// TwinCAT 3 PLC project SYNC
// ProgramVersion: 3.1.4022.2
// libraries:
//   Tc2_EtherCAT, * (Beckhoff Automation GmbH)
//   Tc2_MC2, * (Beckhoff Automation GmbH)
//   Tc2_MC2_Camming, * (Beckhoff Automation GmbH)
//   Tc2_MC2_XFC, * (Beckhoff Automation GmbH)
//   Tc2_Standard, * (Beckhoff Automation GmbH)
//   Tc2_System, * (Beckhoff Automation GmbH)
//   Tc3_Module, * (Beckhoff Automation GmbH)
// project tree:
//   / Plc_Task_SYNC.TcTTO
//   POUs/ AxisController.TcPOU, BlockerController.TcPOU, CamInController.TcPOU, MAIN.TcPOU, MODULO.TcPOU
// (motion and I/O tree: see PLC project clock)
// real-time tasks:
//   TASK Plc_Task_CLOCK: cycle T#1ms, priority 20, ADS port 350
//   TASK Plc_Task_SYNC: cycle T#10ms, priority 21, ADS port 351
// variable links:
//   CLOCK Instance <-> SYNC/SYNC Instance
//     PlcTask Outputs/MAIN.tPulse <-> Plc_Task_SYNC Inputs/MAIN.tPulse

CONFIGURATION SYNC
    RESOURCE PLC ON TwinCAT3
        TASK Plc_Task_SYNC(INTERVAL := T#10ms, PRIORITY := 21);
        PROGRAM MAIN WITH Plc_Task_SYNC : MAIN;
    END_RESOURCE
END_CONFIGURATION

// ---- POUs/MAIN.TcPOU
PROGRAM MAIN
VAR
	
	tPulse AT %I*: T_DCTIME64;
	tPrev : T_DCTIME64;
	tPrevPulse : T_DCTIME64;
	tDiff : T_DCTIME64;
	
	SyncMaster : AXIS_REF;
	SyncSlave : AXIS_REF;

	XFC_Position : XFC_PositionAtTime;
	
	fPosition : LREAL;
	fPositionMod : LREAL;
	fPrevPosition : LREAL;
	
	fPositionError : LREAL;
	fPositionSum : LREAL;
	
	fSpeedError : LREAL;
	fSpeedAct : LREAL;
	fSpeed : LREAL := 360*14;
	
	fPositionDiff : LREAL;
	
	Master : AxisController;
	Slave : CamInController;
	
	mcMoveVelo : MC_MoveVelocity;
	
	iState : UINT;
	bPulse : BOOL;
	
	fSpeed_Kp : LREAL := 0.1;
	
	fPosition_Kp : LREAL := 0.1;
	fPosition_Ki : LREAL := 0.001;
	
	fPositionControlThreshold: LREAL := 10;
	
END_VAR

Master(Axis:=SyncMaster);
Master.bExecute:=FALSE;

Slave(Axis:=SyncSlave, Master:=SyncMaster);
Slave.bExecute:=FALSE;

mcMoveVelo(Axis:=SyncMaster);
mcMoveVelo.Execute := FALSE;

CASE iState OF
	000:
		// Compose a camming table?
		
		iState := 100;

	100:
		// Set up the master axis
		Master.fSpeed:=0;
		Master.bExecute := TRUE;
		iState := 101;
	101:
		IF Master.bDone THEN
			iState:= 200;
		END_IF
		
	200:
		// Check for new pulse
		IF tPulse <> tPrev THEN
			// There's a new pusle
			fPrevPosition := fPosition;
			tPrevPulse := tPrev;
			bPulse := TRUE;
		
			// Get the position at the pulse
			XFC_Position(DcTime:=ULINT_TO_UDINT(tPulse), Axis:= SyncMaster);
			fPosition := XFC_Position.Position;
			fPositionMod := MODULO(XFC_Position.Position+180, 360)-180;
			
			// Calculate the distance moved
			fPositionDiff := fPosition-fPrevPosition;
			
			// Calculate the time between pulses
			tDiff := tPulse - tPrevPulse;
			
			// Calculate the actual speed
			fSpeedAct := fPositionDiff/tDiff*1E9;
			
			// Calculate the speed difference - with respect to the expected 360degrees
			fSpeedError := -(fPositionDiff-360)/tDiff*1E9;
			
			// Implement the speed PI controller
			fSpeed := fSpeed + fSpeedError*fSpeed_Kp;
			
			// Implement the position PI controller
			fPositionError := MODULO(fPosition+180, 360)-180;
			fPositionSum := fPositionSum + fPositionError;
			
			// Only activate position control if the speed control is good
			IF ABS(fSpeedError) < fPositionControlThreshold THEN
				fSpeed := fSpeed - fPositionError * fPosition_Kp;
				fSpeed := fSpeed - fPositionSum * fPosition_Ki;
			ELSE
				fPositionSum := 0;
			END_IF
			
			IF fSpeed > 5700 THEN
				fSpeed := 5700;
			END_IF
			
			// Update the velocity
			mcMoveVelo.Execute:= TRUE;
			mcMoveVelo.Velocity:= fSpeed;
			
			(*// Activate slave camming?
			IF NOT Slave.bDone THEN
				Slave.bExecute:=TRUE;
			END_IF*)
		
		ELSE
			bPulse := FALSE;
		END_IF
		
		tPrev := tPulse;
			
END_CASE

END_PROGRAM

// ---- POUs/AxisController.TcPOU
FUNCTION_BLOCK AxisController
VAR_INPUT
	bExecute: BOOL;
	fSpeed : LREAL := 360;
END_VAR
VAR
	mcReset			: MC_Reset;
	mcPower			: MC_Power;
	mcMoveVelo		: MC_MoveVelocity;
	mcStop			: MC_Stop;
	
	iState: UINT;;
END_VAR
VAR_IN_OUT
	Axis : AXIS_REF;
END_VAR
VAR_OUTPUT
	bDone : BOOL;
END_VAR

mcReset(Axis:=Axis);
mcReset.Execute := FALSE;

mcPower(Axis:=Axis, Enable:=TRUE, Enable_Positive:=TRUE, Enable_Negative:=TRUE);

mcMoveVelo(Axis:=Axis);
mcMoveVelo.Execute := FALSE;

CASE iState OF
	0:		
		IF bExecute THEN
			iState:= 10;
		END_IF
		
	10: 
		// Reset the axis
		mcReset.Execute:=TRUE;
		iState := 20;
		bDone:= FALSE;
	
	20: 
		// Wait for reset to complete
		IF McReset.Done THEN
			iState := 30;
		ELSIF McReset.Error THEN
			iState := 999;
		END_IF
	
	30:
		// Set the power!
		IF McPower.Status THEN
			iState := 40;
		END_IF
		
	40: 
		// Move at constant velo
		mcMoveVelo.Execute := TRUE;
		mcMoveVelo.Velocity:=fSpeed;
		
		iState:= 50;
	
	50: 
		// Done.
		IF mcMoveVelo.InVelocity THEN
			bDone := TRUE;
			iState := 0;
		END_IF
		
END_CASE

END_FUNCTION_BLOCK

// ---- POUs/CamInController.TcPOU
FUNCTION_BLOCK CamInController
VAR_INPUT
	bExecute: BOOL;
	fSpeed : LREAL := 360;
END_VAR
VAR
	mcReset			: MC_Reset;
	mcPower			: MC_Power;
	mcStop			: MC_Stop;
	mcCamIn         : MC_CamIn;
	
	iState: UINT;;
END_VAR
VAR_IN_OUT
	Axis : AXIS_REF;
	Master : AXIS_REF;
END_VAR
VAR_OUTPUT
	bDone : BOOL;
END_VAR

mcReset(Axis:=Axis);
mcReset.Execute := FALSE;

mcPower(Axis:=Axis, Enable:=TRUE, Enable_Positive:=TRUE, Enable_Negative:=TRUE);

mcCamIn(Slave:=Axis, Master:= Master);
mcCamIn.Execute:=FALSE;

CASE iState OF
	0:	
		IF bExecute THEN
			iState:= 10;
		END_IF
		
	10: 
		// Reset the axis
		mcReset.Execute:=TRUE;
		iState := 20;
		bDone:= FALSE;
	
	20: 
		// Wait for reset to complete
		IF McReset.Done THEN
			iState := 30;
		ELSIF McReset.Error THEN
			iState := 999;
		END_IF
	
	30:
		// Set the power!
		IF McPower.Status THEN
			iState := 40;
		END_IF
		
	40:
		// Cam in
		mcCamIn.Execute:= TRUE;
		mcCamIn.SlaveScaling:= 1; 
		mcCamIn.CamTableID:= 1;
		
		iState:= 50;
	
	50: 
		// Done.
		IF mcCamIn.InSync THEN
			bDone := TRUE;
			iState := 0;
		END_IF
		
END_CASE

END_FUNCTION_BLOCK

// ---- POUs/MODULO.TcPOU
FUNCTION MODULO : LREAL
VAR_INPUT
	fValue : LREAL;
	fDenom : LREAL := 360;
END_VAR
VAR
END_VAR

MODULO := fValue - (TRUNC(fValue / fDenom) * fDenom);

END_FUNCTION

// ---- POUs/BlockerController.TcPOU
FUNCTION_BLOCK BlockerController
VAR_INPUT
	bExecute: BOOL;
	fSpeed : LREAL := 360;
	
	bPulse : BOOL;
	
	iHi : UINT := 1;
	iLo : UINT := 1;
END_VAR
VAR
	mcReset			: MC_Reset;
	mcPower			: MC_Power;
	mcStop			: MC_Stop;
	mcCamIn         : MC_CamIn;
	mcCamOut		: MC_CamOut;
	
	stCamInOptions  : ST_CamInOptions;
	stCamOutOptions : ST_CamOutOptions;
	
	iState: UINT;
	
	iCounter : UINT;
END_VAR
VAR_IN_OUT
	Axis : AXIS_REF;
	Master : AXIS_REF;
END_VAR
VAR_OUTPUT
	bRunning : BOOL;
END_VAR

mcReset(Axis:=Axis);
mcReset.Execute := FALSE;

mcPower(Axis:=Axis, Enable:=TRUE, Enable_Positive:=TRUE, Enable_Negative:=TRUE);

mcCamIn(Slave:=Axis, Master:= Master, Options:= stCamInOptions);
mcCamIn.Execute:=FALSE;

mcCamOut(Slave:=Axis, Options:= stCamOutOptions);
mcCamOut.Execute:=FALSE;

CASE iState OF
	0:	
		IF bExecute THEN
			iState:= 10;
		END_IF
		bRunning := FALSE;
		
	10: 
		// Reset the axis
		mcReset.Execute:=TRUE;
		iState := 20;
	
	20: 
		// Wait for reset to complete
		IF McReset.Done THEN
			iState := 30;
		ELSIF McReset.Error THEN
			iState := 999;
		END_IF
	
	30:
		// Set the power!
		IF McPower.Status THEN
			iState := 40;
			bRunning := TRUE;
		END_IF
		
	40:
		// Cam in
		mcCamIn.Execute:= TRUE;
		mcCamIn.SlaveScaling:= 1; 
		mcCamIn.CamTableID:= 1;
		
		stCamInOptions.ActivationMode:= MC_CAMACTIVATION_NEXTCYCLE;
		
		iState:= 50;
	
	50: 
		// Cam out
		IF mcCamIn.InSync THEN
			mcCamOut.Execute:=TRUE;
			iState := 60;
		END_IF
		
	60:
		// Count pulses
		IF bPulse THEN
			iCounter := iCounter + 1;
		END_IF
		
		// Check if hi pulse count reached
		IF iCounter < iHi THEN
			iCounter := 0;
			
			iState:= 70;
		END_IF
		
		
END_CASE

END_FUNCTION_BLOCK
